RoboDK station: Simulation & programs.rdk

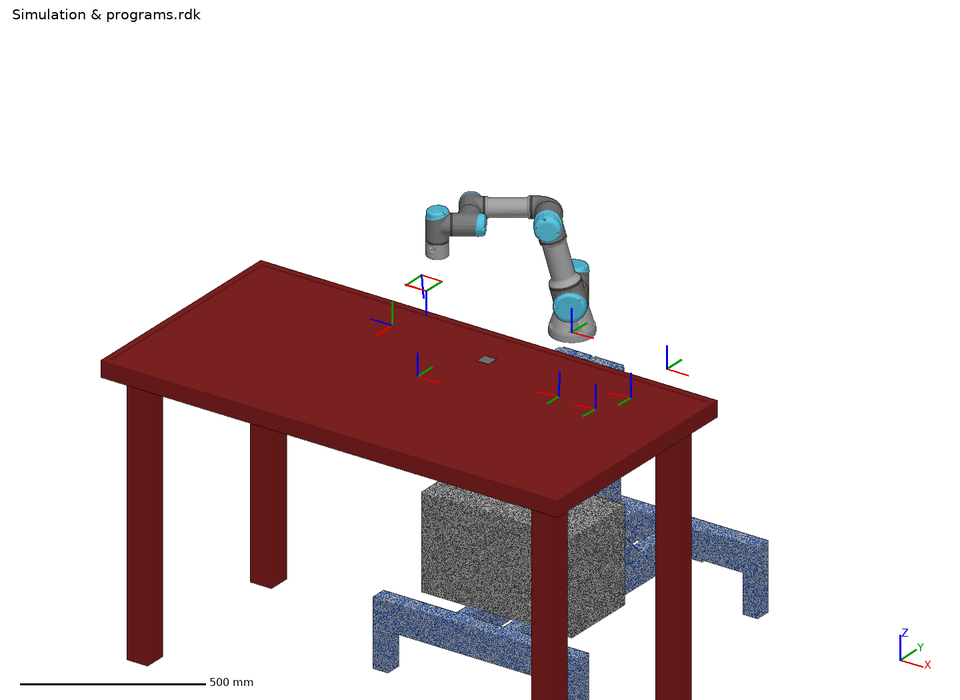
[picture v0: the station drawn from its stored meshes, robots at their saved joint values, targets as dots, program paths as lines]
Station Simulacion_3e (saved by RoboDK 5.6.3). Poses are relative to the parent item; angles as X-Y-Z fixed-axis rotations.
Station parameters (name, value as stored): RECORD_READY, 1, RECORD_STOP, 0, RECORD_ACKNOWLEDGE, 1, RECORD_ROBOT, 1
  - frame UR3e Base at (0, 0, 0) mm
    - robot UR3e: 6 axes, payload 3 kg, reach 500 mm, repeatability 0.03 mm, weight 11 kg
        modified DH rows (alpha deg, a mm, theta deg, d mm): 0, 0, 0, 151.9; 90, 0, 180, 0; 0, 243.55, 0, 0; 0, 213.2, 0, 131.05; -90, 0, 0, 85.35; 90, 0, 180, 92.1
        joint limits [-360, -360, -360, -360, -360, -360] to [360, 360, 360, 360, 360, 360]; home [90, -90, 90, -90, -90, 0]; saved at [32.842, -75.693, 77.295, -91.601, -89.995, -57.158]
      - frame Frame_Camara_1 at (9.13, -59.06, 41.13) mm, rotated rx 2.97 ry 2.34 rz -176.88 deg
        - camera CamaraBrazo
      - tool Gripper 2, TCP at (0, -50, 90) mm
      - frame Frame 8 at (0, -50, 90) mm
    - frame huevo_0 at (365.18, -244.95, 4.03) mm, rotated rx 5.66 ry 2.48 rz -173.5 deg
    - frame huevo_1 at (340.38, -375.16, 14.87) mm, rotated rx 5.66 ry 2.48 rz -173.5 deg
    - frame huevo_2 at (204.36, -351.92, 5.32) mm, rotated rx 5.66 ry 2.48 rz -173.5 deg
  - object mesaUR v1 at (0, 0, -110) mm, rotated rx 0 ry 0 rz -90 deg, size 1282 x 1503 x 903.8 mm
  - frame Frame_Tablero at (-200.86, -439.4, -14.21) mm
    - object Checkerboard at (0, 0, 0) mm, size 148.6 x 105 x 0 mm, geometry from Checkerboard.png
  - frame Frame_Aruco_20 at (340, -40, 0) mm
    - object aruco-20 at (-450, -250, 0) mm, size 37.9 x 37.9 x 0 mm, geometry from aruco-20.png
  - object Huevo at (-87.8, -330.3, 0) mm, rotated rx 0 ry 0 rz 60 deg, size 44.9 x 57 x 45 mm, geometry from Huevo.STEP
  - object Huevo at (10, -320, 0) mm, rotated rx 0 ry 0 rz 140 deg, size 44.9 x 57 x 45 mm, geometry from Huevo.STEP
  - object Huevo at (400, -90, 0) mm, rotated rx 0 ry 0 rz -15 deg, size 44.9 x 57 x 45 mm, geometry from Huevo.STEP
  - Python program Hand-Eye acquisition (listed below)
  - Python program Hand-Eye calibration (listed below)
  - Python program Hand-Eye acquisition Aruco (listed below)
  - Python program Tomar Una Foto (listed below)
  - Python program Pos (listed below)
  - frame PrePallet at (-230.35, -354.58, 199.88) mm, rotated rx -179.99 ry 0 rz 179.99 deg
  - Python program USB (listed below)
  - Python program TestMQTT (listed below)
  - frame inicioPallet at (-350.36, -344.58, 59.9) mm, rotated rx 90 ry 0 rz -90 deg
  - Python program Pos2 (listed below)

--- Python program Hand-Eye acquisition ---
# Type help("robolink") or help("robodk") for more information
# Press F5 to run the script
# Documentation: https://robodk.com/doc/en/RoboDK-API.html
# Reference:     https://robodk.com/doc/en/PythonAPI/index.html
#
# Utility script to perform hand-eye calibration on a 2D camera.
# This script can be use for eye-in-hand or eye-to-hand calibrations.
# Dynamically record the robot pose and save the camera image on disk for later processing.
# This script is running in a separate thread and a main program request punctual recordings through an handshake.

from robodk import robolink  # RoboDK API
from robodk import robomath  # Robot toolbox

# Uncomment these lines to automatically install the dependencies using pip
# robolink.import_install('cv2', 'opencv-contrib-python==4.5.*')
# robolink.import_install('numpy')
import cv2 as cv
import numpy as np
from pathlib import Path
import json
from enum import Enum
import time


#--------------------------------------
# This script supports RoboDK virtual/simulated cameras, and USB devices (as supported by OpenCV)
# You can add your own implementation to retrieve images from any camera, such as a Cognex Insight, SICK, etc.
class CameraTypes(Enum):
    ROBODK_SIMULATED = 1
    OPENCV_USB = 0


RECORD_ROBOT = True  # Record the robot pose on disk
RECORD_CAMERA = True  # Record the camera image on disk
RECORD_FOLDER = 'Calibracion Hand - Eye Camara'  # Default folder to save recordings, relative to the station folder

CAMERA_TYPE = CameraTypes.OPENCV_USB  # Camera type to be used
CAMERA_ROBODK_NAME = 'My Camera'  # [Optional] Default name to use for the RoboDK camera
ROBOT_NAME = 'UR3e'  # [Optional] Default name to use for the robot

# Station variables shared with the main program to interact with this script
RECORD_READY = 'RECORD_READY'  # Set this true in the main program when the robot is in position and the the script is allowed to record the robot and the image
RECORD_ACKNOWLEDGE = 'RECORD_ACKNOWLEDGE'  # Set this true in this script when the record is complete
RECORD_STOP = 'RECORD_STOP'  # Request to stop the script by the main program


#--------------------------------------
def get_robot(RDK: robolink.Robolink, robot_name: str):

    # Retrieve the robot
    robot_item = None
    if robot_name:
        robot_item = RDK.Item(robot_name, robolink.ITEM_TYPE_ROBOT)
        if not robot_item.Valid():
            robot_name = ''

    if not robot_name:
        robot_item = RDK.ItemUserPick("Select the robot for hand-eye", robolink.ITEM_TYPE_ROBOT)
        if not robot_item.Valid():
            raise

    return robot_item


def get_camera_handle(camera_type: CameraTypes, camera_name: str, RDK: robolink.Robolink):

    if camera_type == CameraTypes.ROBODK_SIMULATED:

        # Retrieve the RoboDK camera by name
        camera_item = None
        if camera_name:
            camera_item = RDK.Item(camera_name, robolink.ITEM_TYPE_CAMERA)
            if not camera_item.Valid():
                camera_name = ''

        if not camera_name:
            camera_item = RDK.ItemUserPick("Select the camera for hand-eye", robolink.ITEM_TYPE_CAMERA)
            if not camera_item.Valid():
                raise

        # Ensure the preview window in RoboDK is open
        if camera_item.setParam('Open') != '1':
            camera_item.setParam('Open', 1)
            robomath.pause(0.1)

        return camera_item

    elif camera_type == CameraTypes.OPENCV_USB:
        return cv.VideoCapture(0, cv.CAP_ANY)  # More information on supported devices here: https://docs.opencv.org/4.x/d8/dfe/classcv_1_1VideoCapture.html#aabce0d83aa0da9af802455e8cf5fd181

    return None


def record_camera(camera_type: CameraTypes, camera_handle, filename: str):
    if camera_type == CameraTypes.ROBODK_SIMULATED:
        record_robodk_camera(filename, camera_handle)

    elif camera_type == CameraTypes.OPENCV_USB:
        record_opencv_camera(filename, camera_handle)


def record_robodk_camera(filename: str, camera_item: robolink.Item):

    # Retrieve the image by socket
    bytes_img = camera_item.RDK().Cam2D_Snapshot('', camera_item)
    nparr = np.frombuffer(bytes_img, np.uint8)
    img = cv.imdecode(nparr, cv.IMREAD_COLOR)

    # Save the image on disk as a grayscale image
    cv.imwrite(filename, cv.cvtColor(img, cv.COLOR_RGB2GRAY))


def record_opencv_camera(filename: str, capture: cv.VideoCapture(0)):

    capture.set(3, 1280)  # Ancho
    capture.set(4, 720)

    # Retrieve image
    success, img = capture.read()
    if not success:
        raise



    # Save the image on disk as a grayscale image
    cv.imwrite(filename, cv.cvtColor(img, cv.COLOR_RGB2GRAY))


def record_robot(robot_item: robolink.Item, filename: str):

    # Retrieve the required information for hand-eye
    robot_data = {}
    robot_data['joints'] = robot_item.Joints().tolist()
    robot_data['pose_flange'] = robomath.Pose_2_TxyzRxyz(robot_item.SolveFK(robot_item.Joints()))

    # Save it on disk as a JSON
    # You can also provide another format, like YAML
    with open(filename, 'w') as f:
        json.dump(robot_data, f, indent=2)


def runmain():

    RDK = robolink.Robolink()

    # Retrieve the camera and robot
    camera_handle = get_camera_handle(CAMERA_TYPE, CAMERA_ROBODK_NAME, RDK)
    #print ("Camera name:" + camera_handle.Name())
    robot_item = get_robot(RDK, ROBOT_NAME)
    #print ("Robot name:" + robot_item.Name())

    # Retrieve the folder to save the data
    record_folder = Path(RDK.getParam(robolink.PATH_OPENSTATION)) / RECORD_FOLDER
    record_folder.mkdir(exist_ok=True, parents=True)
    print ("Folder ok")
    # This script does not delete the previous run if the folder is not empty
    # If the folder is not empty, retrieve the next ID
    id = 0
    ids = sorted([int(x.stem) for x in record_folder.glob('*.png') if x.stem.isdigit()])
    if ids:
        id = ids[-1] + 1

    # Start the main loop, and wait for requests
    RDK.setParam(RECORD_READY, 0)
    while True:
        time.sleep(0.01)

        # Read the requests set by the main program
        ready = int(RDK.getParam(RECORD_READY)) == 1
        stop = int(RDK.getParam(RECORD_STOP)) == 1
        if stop:

            break

        if not ready:

            continue



        # Process the requests
        if RECORD_CAMERA:
            img_filename = Path(f'{record_folder.as_posix()}/{id}.png')
            record_camera(CAMERA_TYPE, camera_handle, img_filename.as_posix())

        if RECORD_ROBOT:
            robot_filename = Path(f'{record_folder.as_posix()}/{id}.json')
            record_robot(robot_item, robot_filename.as_posix())

        id += 1

        print(img_filename)
        print(robot_filename)

        # Inform the main program that we have completed the request
        RDK.setParam(RECORD_ACKNOWLEDGE, 1)
        RDK.setParam(RECORD_READY, 0)




if __name__ == '__main__':
    runmain()

--- Python program Hand-Eye calibration ---
# Type help("robolink") or help("robodk") for more information
# Press F5 to run the script
# Documentation: https://robodk.com/doc/en/RoboDK-API.html
# Reference:     https://robodk.com/doc/en/PythonAPI/index.html
#
# Perform hand-eye calibration with recorded robot poses and 2D images from disk.
# - Requires at least 8 different poses at different orientations/distances of a chessboard or charucoboard.
# - Requires a calibrated camera (known intrinsic parameters, including distortion), which can also be performed from local images.
#
# You can find the board used in this example here:
# https://docs.opencv.org/4.x/charucoboard.png
#

from robodk import robolink  # RoboDK API
from robodk import robomath  # Robot toolbox
from robodk import robodialogs  # Dialogs

# Uncomment these lines to automatically install the dependencies using pip
# robolink.import_install('cv2', 'opencv-contrib-python==4.5.*')
# robolink.import_install('numpy')
import cv2 as cv
import numpy as np
import json
from pathlib import Path
from enum import Enum


#--------------------------------------
# This scripts supports chessboard (checkerboard) and ChAruCo board as calibration objects.
# You can add your own implementation (such as dot patterns).
class MarkerTypes(Enum):
    CHESSBOARD = 0
    CHARUCOBOARD = 1


# The camera intrinsic parameters can be performed with the same board as the Hand-eye
INTRINSIC_FOLDER = 'B:/Descargas/Simulacion 3e/Simulacion 3e/Calibracion Hand - Eye Camara'  # Default folder to load images for the camera calibration, relative to the station folder
HANDEYE_FOLDER = 'B:/Descargas/Simulacion 3e/Simulacion 3e/Calibracion Hand - Eye Camara'
# Camera intrinsic calibration board parameters
# You can find this chessboard here: https://docs.opencv.org/4.x/charucoboard.png
INTRINSIC_BOARD_TYPE = MarkerTypes.CHESSBOARD
INTRINSIC_CHESS_SIZE = (11, 9)  # X/Y
INTRINSIC_SQUARE_SIZE = 18  # mm
INTRINSIC_MARKER_SIZE = 18 # mm

# Hand-eye calibration board parameters
# You can find this charucoboard here: https://docs.opencv.org/4.x/charucoboard.png
#HANDEYE_BOARD_TYPE = MarkerTypes.CHARUCOBOARD
HANDEYE_BOARD_TYPE = MarkerTypes.CHESSBOARD
HANDEYE_CHESS_SIZE = (11, 9)  # X/Y
HANDEYE_SQUARE_SIZE = 18 # mm
HANDEYE_MARKER_SIZE = 18 # mm


def pose_2_Rt(pose: robomath.Mat):
    """RoboDK pose to OpenCV pose"""
    pose_inv = pose.inv()
    R = np.array(pose_inv.Rot33())
    t = np.array(pose.Pos())
    return R, t


def Rt_2_pose(R, t):
    """OpenCV pose to RoboDK pose"""
    vx, vy, vz = R.tolist()

    cam_pose = robomath.eye(4)
    cam_pose.setPos([0, 0, 0])
    cam_pose.setVX(vx)
    cam_pose.setVY(vy)
    cam_pose.setVZ(vz)

    pose = cam_pose.inv()
    pose.setPos(t.tolist())

    return pose


def find_chessboard(img, mtx, dist, chess_size, squares_edge, refine=True, draw_img=None):
    """
    Detects a chessboard pattern in an image.
    """

    pattern = np.subtract(chess_size, (1, 1))  # number of corners

    # Prefer grayscale images
    _img = img
    if len(img.shape) > 2:
        _img = cv.cvtColor(img, cv.COLOR_RGB2GRAY)

    # Find the chessboard's corners
    success, corners = cv.findChessboardCorners(_img, pattern)
    if not success:
        raise Exception("No chessboard found")

    # Refine
    if refine:
        criteria = (cv.TERM_CRITERIA_EPS + cv.TERM_CRITERIA_MAX_ITER, 30, 0.001)
        search_size = (11, 11)
        zero_size = (-1, -1)
        corners = cv.cornerSubPix(_img, corners, search_size, zero_size, criteria)

    if draw_img is not None:
        cv.drawChessboardCorners(draw_img, pattern, corners, success)

    # Find the camera pose. Only available with the camera matrix!
    if mtx is None or dist is None:
        return corners, None, None

    cb_corners = np.zeros((pattern[0] * pattern[1], 3), np.float32)
    cb_corners[:, :2] = np.mgrid[0:pattern[0], 0:pattern[1]].T.reshape(-1, 2) * squares_edge
    success, rvec, tvec = cv.solvePnP(cb_corners, corners, mtx, dist)
    if not success:
        raise Exception("No chessboard found")

    R_target2cam = cv.Rodrigues(rvec)[0]
    t_target2cam = tvec

    return corners, R_target2cam, t_target2cam


def find_charucoboard(img, mtx, dist, chess_size, squares_edge, markers_edge, predefined_dict=cv.aruco.DICT_6X6_100, draw_img=None) -> dict:
    """
    Detects a charuco board pattern in an image.
    """

    # Note that for chessboards, the pattern size is the number of "inner corners", while charucoboards are the number of chessboard squares

    # Charuco board and dictionary
    charuco_board = cv.aruco.CharucoBoard_create(chess_size[0], chess_size[1], squares_edge, markers_edge, cv.aruco.getPredefinedDictionary(predefined_dict))
    charuco_dict = charuco_board.dictionary

    # Find the markers first
    marker_corners, marker_ids, _ = cv.aruco.detectMarkers(img, charuco_dict, None, None, None, None)
    if marker_ids is None or len(marker_ids) < 1:
        raise Exception("No charucoboard found")

    # Then the charuco
    count, corners, ids = cv.aruco.interpolateCornersCharuco(marker_corners, marker_ids, img, charuco_board, None, None, mtx, dist, 2)  # mtx and dist are optional here
    if count < 1 or len(ids) < 1:
        raise Exception("No charucoboard found")

    if draw_img is not None:
        cv.aruco.drawDetectedCornersCharuco(draw_img, corners, ids)

    # Find the camera pose. Only available with the camera matrix!
    if mtx is None or dist is None:
        return corners, None, None

    success, rot_vec, trans_vec = cv.aruco.estimatePoseCharucoBoard(corners, ids, charuco_board, mtx, dist, None, None, False)  # mtx and dist are mandatory here
    if not success:
        raise Exception("Charucoboard pose not found")

    if draw_img is not None:
        cv.drawFrameAxes(draw_img, mtx, dist, rot_vec, trans_vec, max(1.5 * squares_edge, 5))

    R_target2cam = cv.Rodrigues(rot_vec)[0]

    return corners, R_target2cam, trans_vec


def calibrate_static(chessboard_images, board_type: MarkerTypes, chess_size, squares_edge: float, markers_edge: float, min_detect: int = -1, show_images=False):
    """
    Calibrate a camera with a chessboard or charucoboard pattern.
    """
    # Chessboard parameters
    pattern = np.subtract(chess_size, (1, 1))  # number of corners
    img_size = None

    # Find the chessboard corners
    img_corners = []

    if show_images:
        WDW_NAME = 'Chessboard'
        MAX_W, MAX_H = 640, 480
        cv.namedWindow(WDW_NAME, cv.WINDOW_NORMAL)

    for file, img in chessboard_images.items():
        # Ensure the image size is consistent
        if img_size is None:
            img_size = img.shape[:2]
        else:
            if img.shape[:2] != img_size:
                raise Exception('Camera resolution is not consistent across images!')

        # Find the chessboard corners
        draw_img = None
        if show_images:
            draw_img = cv.cvtColor(img, cv.COLOR_GRAY2RGB)
        try:
            if board_type == MarkerTypes.CHESSBOARD:
                corners, _, _ = find_chessboard(img, mtx=None, dist=None, chess_size=chess_size, squares_edge=squares_edge, draw_img=draw_img)
            else:
                corners, _, _ = find_charucoboard(img, mtx=None, dist=None, chess_size=chess_size, squares_edge=squares_edge, markers_edge=markers_edge, draw_img=draw_img)
        except:
            print(f'Unable to find chessboard in {file}!')
            continue

        if show_images:
            cv.imshow(WDW_NAME, draw_img)
            cv.resizeWindow(WDW_NAME, MAX_W, MAX_H)
            cv.waitKey(500)
        img_corners.append(corners)

        # Check if we processed enough images
        if min_detect > 0 and len(img_corners) >= min_detect:
            break

    if show_images:
        cv.destroyAllWindows()

    if len(img_corners) < 3 or min_detect > 0 and len(img_corners) < min_detect:
        raise Exception('Not enough detections!')

    # Calibrate the camera
    # Create a flat chessboard representation of the corners
    cb_corners = np.zeros((pattern[0] * pattern[1], 3), np.float32)
    cb_corners[:, :2] = np.mgrid[0:pattern[0], 0:pattern[1]].T.reshape(-1, 2) * squares_edge

    h, w = img_size
    rms_err, mtx, dist, rot_vecs, trans_vecs = cv.calibrateCamera([cb_corners for i in range(len(img_corners))], img_corners, (w, h), None, None)
    return mtx, dist, (w, h)


def calibrate_handeye(robot_poses, chessboard_images, camera_matrix, camera_distortion, board_type: MarkerTypes, chess_size, squares_edge: float, markers_edge: float, show_images=False):
    """
    Calibrate a camera mounted on a robot arm using a list of robot poses and a list of images for each pose.
    The robot pose should be at the flange (remove .PoseTool) unless you have a calibrated tool.
    """
    # https://docs.opencv.org/4.x/d9/d0c/group__calib3d.html#gaebfc1c9f7434196a374c382abf43439b

    # Rotation part extracted from the homogeneous matrix that transforms a point expressed in the gripper frame to the robot base frame (bTg).
    # This is a vector (vector<Mat>) that contains the rotation, (3x3) rotation matrices or (3x1) rotation vectors, for all the transformations from gripper frame to robot base frame.
    R_gripper2base_list = []

    # Translation part extracted from the homogeneous matrix that transforms a point expressed in the gripper frame to the robot base frame (bTg).
    # This is a vector (vector<Mat>) that contains the (3x1) translation vectors for all the transformations from gripper frame to robot base frame.
    t_gripper2base_list = []

    # Rotation part extracted from the homogeneous matrix that transforms a point expressed in the target frame to the camera frame (cTt).
    # This is a vector (vector<Mat>) that contains the rotation, (3x3) rotation matrices or (3x1) rotation vectors, for all the transformations from calibration target frame to camera frame.
    R_target2cam_list = []

    # Rotation part extracted from the homogeneous matrix that transforms a point expressed in the target frame to the camera frame (cTt).
    # This is a vector (vector<Mat>) that contains the (3x1) translation vectors for all the transformations from calibration target frame to camera frame.
    t_target2cam_list = []

    if show_images:
        WDW_NAME = 'Charucoboard'
        #WDW_NAME = 'Chessboard'
        MAX_W, MAX_H = 640, 480
        cv.namedWindow(WDW_NAME, cv.WINDOW_NORMAL)

    for i in chessboard_images.keys():
        robot_pose = robot_poses[i]
        image = chessboard_images[i]
        draw_img = None
        if show_images:
            draw_img = cv.cvtColor(image, cv.COLOR_GRAY2RGB)
        try:
            if board_type == MarkerTypes.CHESSBOARD:
                _, R_target2cam, t_target2cam = find_chessboard(image, camera_matrix, camera_distortion, chess_size, squares_edge, draw_img=draw_img)
            else:
                _, R_target2cam, t_target2cam = find_charucoboard(image, camera_matrix, camera_distortion, chess_size, squares_edge, markers_edge, draw_img=draw_img)
        except:
            print(f'Unable to find chessboard in {i}!')
            continue

        if show_images:
            cv.imshow(WDW_NAME, draw_img)
            cv.resizeWindow(WDW_NAME, MAX_W, MAX_H)
            cv.waitKey(500)

        R_target2cam_list.append(R_target2cam)
        t_target2cam_list.append(t_target2cam)

        R_gripper2base, t_gripper2base = pose_2_Rt(robot_pose)
        R_gripper2base_list.append(R_gripper2base)
        t_gripper2base_list.append(t_gripper2base)

    if show_images:
        cv.destroyAllWindows()

    R_cam2gripper, t_cam2gripper = cv.calibrateHandEye(R_gripper2base_list, t_gripper2base_list, R_target2cam_list, t_target2cam_list)
    return Rt_2_pose(R_cam2gripper, t_cam2gripper)


def runmain():
    #------------------------------------------------------
    # Calibrate the camera intrinsic parameters
    # 1. Print a chessboard, measure it using a caliper
    # 2. Mount the camera statically, take a series of images of the chessboard at different distance, orientation, offset, etc.
    # 3. Calibrate the camera using the images (can be done offline)
    #
    #
    # Calibrate the camera location (hand-eye)
    # 4. Create a robot program in RoboDK that moves the robot around a static chessboard at different distance, orientation, offset, etc.
    # 5. At each position, record the robot pose (robot.Pose(), or robot.Joints() even) and take a screenshot with the camera
    # 6. Use the robot poses and the images to calibrate the camera location
    #
    #
    # Good to know
    # - You can retrieve the camera image live with OpenCV using cv.VideoCapture(0, cv.CAP_DSHOW)
    # - You can load/save images with OpenCV using cv.imread(filename) and cv.imwrite(filename, img)
    # - You can save your calibrated camera parameters with JSON, i.e. print(json.dumps({"mtx":mtx, "dist":dist}))
    #
    #------------------------------------------------------

    RDK = robolink.Robolink()

    #------------------------------------------------------
    # Calibrate a camera using local images of chessboards, retrieves the camera intrinsic parameters
    # Get the input folder
    intrinsic_folder = Path(RDK.getParam(robolink.PATH_OPENSTATION)) / INTRINSIC_FOLDER
    if not intrinsic_folder.exists():
        intrinsic_folder = robodialogs.getSaveFolder(intrinsic_folder.as_posix(), 'Select the directory containing the images (.png) for the camera intrinsic calibration')
        if not intrinsic_folder:
            raise
        intrinsic_folder = Path(intrinsic_folder)

    # Retrieve the images
    image_files = sorted(intrinsic_folder.glob('*.png'))
    images = {int(image_file.stem): cv.imread(image_file.as_posix(), cv.IMREAD_GRAYSCALE) for image_file in image_files}

    # Perform the image calibration
    mtx, dist, size = calibrate_static(images, INTRINSIC_BOARD_TYPE, INTRINSIC_CHESS_SIZE, INTRINSIC_SQUARE_SIZE, INTRINSIC_MARKER_SIZE, min_detect=-1)
    print(f'Camera matrix:\n{mtx}\n')
    print(f'Distortion coefficient:\n{dist}\n')
    print(f'Camera resolution:\n{size}\n')

    #------------------------------------------------------
    # Load images and robot poses to calibrate hand-eye camera
    # Get the input folder
    handeye_folder = Path(RDK.getParam(robolink.PATH_OPENSTATION)) / HANDEYE_FOLDER
    if not handeye_folder.exists():
        handeye_folder = robodialogs.getSaveFolder('Select the directory of the images (.png) and robot poses (.json) for hand-eye calibration')
        if not handeye_folder:
            raise
        handeye_folder = Path(handeye_folder)

    # Retrieve the images and robot poses
    image_files = sorted(handeye_folder.glob('*.png'))
    robot_files = sorted(handeye_folder.glob('*.json'))

    images, poses, joints = {}, {}, {}
    for image_file, robot_file in zip(image_files, robot_files):
        if int(image_file.stem) != int(robot_file.stem):
            raise

        id = int(image_file.stem)

        image = cv.imread(image_file.as_posix(), cv.IMREAD_GRAYSCALE)
        images[id] = image

        with open(robot_file.as_posix(), 'r') as f:
            robot_data = json.load(f)
            joints[id] = robot_data['joints']
            poses[id] = robomath.TxyzRxyz_2_Pose(robot_data['pose_flange'])



    # Perform hand-eye calibration
    camera_pose = calibrate_handeye(poses, images, mtx, dist, HANDEYE_BOARD_TYPE, HANDEYE_CHESS_SIZE, HANDEYE_SQUARE_SIZE, HANDEYE_MARKER_SIZE)



    print(f'Camera pose (wrt to the robot flange):\n{camera_pose}')
    F_C = robomath.Pose_2_UR(camera_pose)
    F_C = np.array(F_C)
    F_C = F_C.tolist()
    ruta_F_C = "B:/Descargas/Simulacion 3e/Simulacion 3e/Matriz_F_C.json"


    mtx = mtx.tolist()
    dist = dist.tolist()
    calibracion = {'F_C':F_C, 'mtx':mtx , 'dist':dist}

    with open(ruta_F_C, 'w') as f:
        json.dump(calibracion, f)
    RDK.ShowMessage('Hand-Eye location:\n' + str(camera_pose))












    #------------------------------------------------------
    # In RoboDK, set the camera location wrt to the robot flange at that calibrated hand-eye location (use a .tool)
    tool = RDK.ItemUserPick('Select the "eye" tool to calibrate', RDK.ItemList(robolink.ITEM_TYPE_TOOL))

    if tool.Valid():
        tool.setPoseTool(camera_pose)




if __name__ == '__main__':
    runmain()

--- Python program Hand-Eye acquisition Aruco ---
# Type help("robolink") or help("robodk") for more information
# Press F5 to run the script
# Documentation: https://robodk.com/doc/en/RoboDK-API.html
# Reference:     https://robodk.com/doc/en/PythonAPI/index.html
#
# Utility script to perform hand-eye calibration on a 2D camera.
# This script can be use for eye-in-hand or eye-to-hand calibrations.
# Dynamically record the robot pose and save the camera image on disk for later processing.
# This script is running in a separate thread and a main program request punctual recordings through an handshake.

from robodk import robolink  # RoboDK API
from robodk import robomath  # Robot toolbox

# Uncomment these lines to automatically install the dependencies using pip
# robolink.import_install('cv2', 'opencv-contrib-python==4.5.*')
# robolink.import_install('numpy')
import cv2 as cv
import numpy as np
from pathlib import Path
import json
from enum import Enum
import time


#--------------------------------------
# This script supports RoboDK virtual/simulated cameras, and USB devices (as supported by OpenCV)
# You can add your own implementation to retrieve images from any camera, such as a Cognex Insight, SICK, etc.
class CameraTypes(Enum):
    ROBODK_SIMULATED = 0
    OPENCV_USB = 1


RECORD_ROBOT = True  # Record the robot pose on disk
RECORD_CAMERA = True  # Record the camera image on disk
RECORD_FOLDER = 'Hand-Eye-Data'  # Default folder to save recordings, relative to the station folder

CAMERA_TYPE = CameraTypes.ROBODK_SIMULATED  # Camera type to be used
CAMERA_ROBODK_NAME = 'My Camera'  # [Optional] Default name to use for the RoboDK camera
ROBOT_NAME = 'UR3e'  # [Optional] Default name to use for the robot

# Station variables shared with the main program to interact with this script
RECORD_READY = 'RECORD_READY'  # Set this true in the main program when the robot is in position and the the script is allowed to record the robot and the image
RECORD_ACKNOWLEDGE = 'RECORD_ACKNOWLEDGE'  # Set this true in this script when the record is complete
RECORD_STOP = 'RECORD_STOP'  # Request to stop the script by the main program


#--------------------------------------
def get_robot(RDK: robolink.Robolink, robot_name: str):

    # Retrieve the robot
    robot_item = None
    if robot_name:
        robot_item = RDK.Item(robot_name, robolink.ITEM_TYPE_ROBOT)
        if not robot_item.Valid():
            robot_name = ''

    if not robot_name:
        robot_item = RDK.ItemUserPick("Select the robot for hand-eye", robolink.ITEM_TYPE_ROBOT)
        if not robot_item.Valid():
            raise

    return robot_item


def get_camera_handle(camera_type: CameraTypes, camera_name: str, RDK: robolink.Robolink):

    if camera_type == CameraTypes.ROBODK_SIMULATED:

        # Retrieve the RoboDK camera by name
        camera_item = None
        if camera_name:
            camera_item = RDK.Item(camera_name, robolink.ITEM_TYPE_CAMERA)
            if not camera_item.Valid():
                camera_name = ''

        if not camera_name:
            camera_item = RDK.ItemUserPick("Select the camera for hand-eye", robolink.ITEM_TYPE_CAMERA)
            if not camera_item.Valid():
                raise

        # Ensure the preview window in RoboDK is open
        if camera_item.setParam('Open') != '1':
            camera_item.setParam('Open', 1)
            robomath.pause(0.1)

        return camera_item

    elif camera_type == CameraTypes.OPENCV_USB:
        return cv.VideoCapture(0, cv.CAP_ANY)  # More information on supported devices here: https://docs.opencv.org/4.x/d8/dfe/classcv_1_1VideoCapture.html#aabce0d83aa0da9af802455e8cf5fd181

    return None


def record_camera(camera_type: CameraTypes, camera_handle, filename: str):
    if camera_type == CameraTypes.ROBODK_SIMULATED:
        record_robodk_camera(filename, camera_handle)

    elif camera_type == CameraTypes.OPENCV_USB:
        record_opencv_camera(filename, camera_handle)


def record_robodk_camera(filename: str, camera_item: robolink.Item):

    # Retrieve the image by socket
    bytes_img = camera_item.RDK().Cam2D_Snapshot('', camera_item)
    nparr = np.frombuffer(bytes_img, np.uint8)
    img = cv.imdecode(nparr, cv.IMREAD_COLOR)

    # Save the image on disk as a grayscale image
    cv.imwrite(filename, img)


def record_opencv_camera(filename: str, capture: cv.VideoCapture):

    capture.set(3, 1280)  # Ancho
    capture.set(4, 720)

    # Retrieve image
    success, img = capture.read()
    if not success:
        raise

    # Save the image on disk as a grayscale image
    cv.imwrite(filename, img)


def record_robot(robot_item: robolink.Item, filename: str):

    # Retrieve the required information for hand-eye
    robot_data = {}
    robot_data['joints'] = robot_item.Joints().tolist()
    robot_data['pose_flange'] = robomath.Pose_2_TxyzRxyz(robot_item.SolveFK(robot_item.Joints()))

    # Save it on disk as a JSON
    # You can also provide another format, like YAML
    with open(filename, 'w') as f:
        json.dump(robot_data, f, indent=2)


def runmain():

    RDK = robolink.Robolink()

    # Retrieve the camera and robot
    camera_handle = get_camera_handle(CAMERA_TYPE, CAMERA_ROBODK_NAME, RDK)
    #print ("Camera name:" + camera_handle.Name())
    robot_item = get_robot(RDK, ROBOT_NAME)
    #print ("Robot name:" + robot_item.Name())

    # Retrieve the folder to save the data
    record_folder = Path(RDK.getParam(robolink.PATH_OPENSTATION)) / RECORD_FOLDER
    record_folder.mkdir(exist_ok=True, parents=True)
    print ("Folder ok")
    # This script does not delete the previous run if the folder is not empty
    # If the folder is not empty, retrieve the next ID
    id = 0
    ids = sorted([int(x.stem) for x in record_folder.glob('*.png') if x.stem.isdigit()])
    if ids:
        id = ids[-1] + 1

    # Start the main loop, and wait for requests
    RDK.setParam(RECORD_READY, 0)

    while True:
        time.sleep(0.01)

        # Read the requests set by the main program
        ready = int(RDK.getParam(RECORD_READY)) == 1
        stop = int(RDK.getParam(RECORD_STOP)) == 1
        if stop:
            break

        if not ready:
            continue

        # Process the requests
        if RECORD_CAMERA:
            img_filename = Path(f'{record_folder.as_posix()}/{id}.png')
            record_camera(CAMERA_TYPE, camera_handle, img_filename.as_posix())

        if RECORD_ROBOT:
            robot_filename = Path(f'{record_folder.as_posix()}/{id}.json')
            record_robot(robot_item, robot_filename.as_posix())

        id += 1

        print(img_filename)
        print(robot_filename)

        # Inform the main program that we have completed the request
        RDK.setParam(RECORD_ACKNOWLEDGE, 1)
        RDK.setParam(RECORD_READY, 0)


if __name__ == '__main__':
    runmain()

--- Python program Tomar Una Foto ---
from robodk import robolink
from robodk import robomath
RDK = robolink.Robolink()


from robodk import *
from robolink import *
import numpy as np

pause(2)
RECORD_READY = 'RECORD_READY'
RDK.setParam(RECORD_READY, 1)
pause(5)

--- Python program Pos ---
import cv2 as cv
import cv2.aruco as aruco
import numpy as np
import math
from scipy.spatial.transform import Rotation
from robodk import robolink
from robodk import robomath
RDK = robolink.Robolink()
from robodk import *
from robolink import *
import json
import os
import glob
from robolink import Robolink, ITEM_TYPE_FRAME
import paho.mqtt.client as mqtt

#hola boby

robot = RDK.Item('UR3e')
robot_frame = RDK.Item('UR3e Base')
frame = RDK.Item('Frame_Aruco_12')
frame_camara = RDK.Item('Frame_Camara_1')
gripper_tcp = RDK.Item('Gripper')
frame_inicio_pallet = RDK.Item('PrePallet')
arriba_pallet_inicio = RDK.Item('inicioPallet')
gripper_2 = RDK.Item('Gripper 2')
#robot.setTool(gripper_2)

frame_camara = RDK.Item('Frame_Camara_1')
ruta_F_C = "B:/Descargas/Simulacion 3e/Simulacion 3e/Matriz_F_C.json"
Mapeo_huevos = "B:/Descargas/Simulacion 3e/Simulacion 3e/Mapeo_Huevos.json"

with open(ruta_F_C, 'r') as f:
    calibracion = json.load(f)

with open(Mapeo_huevos, 'r') as f:
    mapeo= json.load(f)

pixeles_huevos = np.array(mapeo)



F_C = calibracion['F_C']
mtx = calibracion['mtx']
dist = calibracion['dist']
mtx = np.array(mtx)
dist = np.array(dist)
F_C = robomath.UR_2_Pose(F_C)


broker_address = "15.44.0.237" # Dirección del servidor MQTT
client = mqtt.Client("Antonio") # Nombre del cliente

global cap
cap = cv.VideoCapture(0)
cap.set(cv.CAP_PROP_FRAME_WIDTH, 1920)
cap.set(cv.CAP_PROP_FRAME_HEIGHT, 1080)










def pnp(corners):
    l = 40
    patron = np.array(
        [[0, l, 0], [l,l, 0], [l, 0, 0], [0, 0, 0]], dtype=np.float32
    )
    rvec_arr = np.empty((0, 3, 1))
    tvec_arr = np.empty((0, 3, 1))
    for esquina in corners:
        _, rvec, tvec = cv.solvePnP(patron, esquina, mtx, dist)
        rvec_arr = np.concatenate((rvec_arr, [rvec]), axis=0)
        tvec_arr = np.concatenate((tvec_arr, [tvec]), axis=0)

    return rvec_arr, tvec_arr

def ordenar_ids(marker_IDs, marker_corners):
        if marker_IDs is not None:
            sorted_indices = np.argsort(marker_IDs, axis=0)
            corners_sorted = np.array(marker_corners)[sorted_indices.flatten()]
            ids_sorted = np.array(marker_IDs)[sorted_indices.flatten()]
            return ids_sorted, corners_sorted
        else:
            return None, None

def promedio(id, aruco):
    caracteristicas_por_id = {}
    for id, caract in zip(id, aruco):
        if id[0] not in caracteristicas_por_id:
            caracteristicas_por_id[id[0]] = []
        caracteristicas_por_id[id[0]].append(caract)

    for id, caract in caracteristicas_por_id.items():
        caract = np.array(caract)
        promedio = np.mean(caract, axis=0)

    return promedio

def CalcularXYZ(u, v, A, rvec, tvec):
    Cord_reales = np.empty((0, 3, 1))

    for rot, tras in zip(rvec, tvec):
        uv = np.float64([[u, v, 1]]).T
        R, _ = cv.Rodrigues(rot)
        Inv_R = np.linalg.inv(R)
        Izda = Inv_R.dot(np.linalg.inv(A).dot(uv))
        Drch = Inv_R.dot(tras)
        s = -45 + Drch[2][0] / Izda[2][0]
        XYZ = Inv_R.dot(s * np.linalg.inv(A).dot(uv) - tras)
        Cord_reales = np.concatenate((Cord_reales, [XYZ]), axis=0)
    return Cord_reales

def medir_angulo_huevo(th):
    contornos , jerarquia = cv.findContours(th , cv.RETR_EXTERNAL , cv.CHAIN_APPROX_NONE)
    if len(contornos) != 0:

        for contorno in contornos:
            momento = cv.moments(contorno)
            if momento["m00"]>170000: #Limita el tamaño de los objetos que detecta
                #print(momento["m00"])
                elipse = cv.fitEllipse(contorno)
                centro , ejes , angulo = elipse

                centro = [int(centro[0]) , int(centro[1])]
                centroP = [centro[0] + 100 , centro[1] + 100]

                longitud = 100
                anguloP = angulo + 90


                x_extremo = int(centro[0] + longitud * np.cos(np.radians(angulo)))
                y_extremo = int(centro[1] + longitud * np.sin(np.radians(angulo)))

                x_1 = int(centro[0] + longitud * np.cos(np.radians(anguloP)))
                y_1 = int(centro[1] + longitud * np.sin(np.radians(anguloP)))

                angulo_horizontal = np.degrees(np.arctan2(y_1 - centro[1], x_1 - centro[0]))
                angulo_horizontal3 = (90 - anguloP) % 360




        return angulo_horizontal3 , centro



def pos_juntas(all_solutions):
    joints = []
    for j in all_solutions:
        conf_RLF = robot.JointsConfig(j).list()
        rear  = conf_RLF[0]
        lower = conf_RLF[1]
        flip  = conf_RLF[2]
        if rear == 1 and lower == 0 and flip == 1:
            joints = j
            break
    return joints
def configuraciones(pose):
    configuraciones = robot.SolveIK_All(pose, robot.PoseTool())
    return configuraciones

def control_angulo_RDK():
    CAM_NAME = 'CamaraBrazo'
    CAM_PARAMS = 'SIZE=1280x720'
    WINDOW_NAME = 'My Camera Feed'
    WINDOW_NAME_BW = 'My Camera BW'


    cam_item = RDK.Item(CAM_NAME, robolink.ITEM_TYPE_CAMERA)
    if not cam_item.Valid():
        cam_item = RDK.Cam2D_Add(RDK.AddFrame(CAM_NAME + ' Frame'), CAM_PARAMS)
        cam_item.setName(CAM_NAME)
    cam_item.setParam('Open', 1)

    angulo_referencia = 360
    while cam_item.setParam('isOpen') == '1':
        img_socket = None
        bytes_img = RDK.Cam2D_Snapshot('', cam_item)
        if isinstance(bytes_img, bytes) and bytes_img != b'':
            nparr = np.frombuffer(bytes_img, np.uint8)
            img_socket = cv.imdecode(nparr, cv.IMREAD_COLOR)
        if img_socket is None:
            break

        grayImage = cv.cvtColor(img_socket, cv.COLOR_BGR2GRAY)
        ret, img_bw = cv.threshold(grayImage, 200, 255, cv.THRESH_BINARY)
        #th = cv.bitwise_not(img_bw)
        angulo, centro  = medir_angulo_huevo(img_bw, img)


        error = angulo-angulo_referencia
        if angulo < 190 or angulo >350:
            #error = 200
            pause(1)
            return('Orientacion correcta')
        else:
            pos_nueva = robot.Pose()*rotz((error*pi/180)*0.2)
            pos_nueva = pos_juntas(configuraciones( pos_nueva))
            robot.MoveJ(pos_nueva)

        key = cv.waitKey(1)
        if key == 27:
            break  # User pressed ESC, exit

    cv.destroyAllWindows()
    RDK.Cam2D_Close(cam_item)

def control_angulo_OPENC_CV():
    angulo_referencia = 360
    while cap:
        ret, frame = cap.read()

        grayImage = cv.cvtColor(frame, cv.COLOR_BGR2GRAY)
        ret, img_bw = cv.threshold(grayImage, 132, 200, cv.THRESH_BINARY)
        #th = cv.bitwise_not(img_bw)
        angulo, centro  = medir_angulo_huevo(img_bw)
        centro1 = [centro[0] + 100 , centro [1] + 100]
        cv.putText(frame, str(angulo), (50, 50), cv.FONT_HERSHEY_SIMPLEX,2, (255, 0, 0), thickness=2)

        cv.imshow("Th" , img_bw)
        cv.imshow("fr" , frame)

        error = angulo-angulo_referencia
        if angulo < 187 or angulo >343:
              return('Orientacion correcta')
        else:
            pos_nueva = robot.Pose()*rotz((error*pi/180)*0.1)
            pos_nueva = pos_juntas(configuraciones( pos_nueva))
            robot.MoveJ(pos_nueva)
            print(angulo)

        if cv.waitKey(1) & 0xFF == ord('q'):
            break
    cap.release()
    cv.destroyAllWindows()


def controlador_posicion_RDK():
    CAM_NAME = 'CamaraBrazo'
    CAM_PARAMS = 'SIZE=1280x720'
    WINDOW_NAME = 'My Camera Feed'
    WINDOW_NAME_BW = 'My Camera BW'


    cam_item = RDK.Item(CAM_NAME, robolink.ITEM_TYPE_CAMERA)
    if not cam_item.Valid():
        cam_item = RDK.Cam2D_Add(RDK.AddFrame(CAM_NAME + ' Frame'), CAM_PARAMS)
        cam_item.setName(CAM_NAME)
    cam_item.setParam('Open', 1)

    centro_referencia = [640, 360]
    centro_referencia = np.array(centro_referencia)
    ganancia = -0.1
    while cam_item.setParam('isOpen') == '1':
        img_socket = None
        bytes_img = RDK.Cam2D_Snapshot('', cam_item)
        if isinstance(bytes_img, bytes) and bytes_img != b'':
            nparr = np.frombuffer(bytes_img, np.uint8)
            img_socket = cv.imdecode(nparr, cv.IMREAD_COLOR)
        if img_socket is None:
            break

        grayImage = cv.cvtColor(img_socket, cv.COLOR_BGR2GRAY)
        ret, img_bw = cv.threshold(grayImage, 200, 255, cv.THRESH_BINARY)
        contornos, r = cv.findContours(img_bw, cv.RETR_TREE, cv.CHAIN_APPROX_SIMPLE)
        #th = cv.bitwise_not(img_bw)
        for contorno in contornos:
            momento = cv.moments(contorno)


            if momento["m00"] > 27000 :
                cx = int(momento["m10"] / momento["m00"])
                cy = int(momento["m01"] / momento["m00"])


        centro = np.array([cx, cy])

        norma = np.linalg.norm(centro_referencia - centro)


        e_x_g = (centro_referencia[0]- cx )*ganancia
        e_y_g = (centro_referencia[1] - cy)*ganancia


        if norma > 20:
            pos_new =robot.Pose()*transl(e_x_g, e_y_g, 0)
            robot.MoveJ(pos_new)



        else:
            pause(1)

            return('1')

        cv.circle(img_socket, (cx, cy), 5, (255, 0,0), -1)
        cv.circle(img_socket, (centro_referencia[0], centro_referencia[1]), 5, (0, 255,0), -1)
        cv.imshow(WINDOW_NAME_BW, img_socket)


        key = cv.waitKey(1)
        if key == 27:
            break  # User pressed ESC, exit

    cv.destroyAllWindows()
    RDK.Cam2D_Close(cam_item)

def control_posicion_OPENC_CV():
    centro_referencia = [911 , 560]
    centro_referencia = np.array(centro_referencia)
    ganancia = 0.009
    while cap:
        ret, frame = cap.read()
        grayImage = cv.cvtColor(frame, cv.COLOR_BGR2GRAY)
        ret, img_bw = cv.threshold(grayImage, 132, 200, cv.THRESH_BINARY)
        cv.circle(frame, (centro_referencia[0], centro_referencia[1]), 5, (0, 255,0), -1)
        cv.circle(img_bw, (centro_referencia[0], centro_referencia[1]), 5, (0, 255,0), -1)
        #th = cv.bitwise_not(img_bw)
        contornos, r = cv.findContours(img_bw, cv.RETR_TREE, cv.CHAIN_APPROX_SIMPLE)
        for contorno in contornos:
            momento = cv.moments(contorno)
            if momento["m00"] > 170000 :
                cx = int(momento["m10"] / momento["m00"])
                cy = int(momento["m01"] / momento["m00"])
                print(cx, cy)
        centro = np.array([cx, cy])
        norma = np.linalg.norm(centro_referencia - centro)
        e_x_g = (centro_referencia[0]- cx )*ganancia
        e_y_g = (centro_referencia[1] - cy)*ganancia
        if norma > 8:
            pos_new =robot.Pose()*transl(e_x_g, e_y_g, 0)
            robot.MoveJ(pos_new)
            print(norma)
            return '1'
        else:
            print('Posicion corregida')
            #return('1')
        cv.circle(frame, (cx, cy), 5, (255, 0,0), -1)
        cv.circle(img_bw, (cx, cy), 5, (255, 0,0), -1)

        cv.imshow('1', frame)
        cv.imshow('2', img_bw)
        if cv.waitKey(1) & 0xFF == ord('q'):
            break
    cap.release()
    cv.destroyAllWindows()

def pallet_size(n, x_p, y_p):
    if n % x_p != 0:
        x = (n // x_p)+1
    else:
        x = n / x_p
    y = []
    for i in range(x):
        if n - y_p > 0:
            y.append(y_p)
        else:
            y.append(n % y_p)
        n = n - y_p
    return x,

def on_message(client, userdata, message):
    global mensaje_global
    mensaje_global = str(message.payload.decode("utf-8"))















ruta_carpeta = "B:/Descargas/Simulacion 3e/Simulacion 3e/Hand-Eye-Data"

archivos_json = sorted(glob.glob(os.path.join(ruta_carpeta, '*.json')))

imagenes = glob.glob(os.path.join(ruta_carpeta, '*.png'))

assert len(archivos_json) == len(imagenes), "La cantidad de archivos .json e imágenes no coincide"
mapa_aruco = np.empty([0,6])
mapa_id = np.empty([0,1])
for archivo_json, img, huevos_pix in zip(archivos_json, imagenes, pixeles_huevos):
    with open(archivo_json, 'r') as f:
        data = json.load(f)

    B_F = data["pose_flange"]
    B_F = robomath.TxyzRxyz_2_Pose(B_F)
    B_F = robomath.Mat(B_F)

    img = cv.imread(img)
    gray_frame = cv.cvtColor(img, cv.COLOR_BGR2GRAY)
    marker_dict = cv.aruco.getPredefinedDictionary(cv.aruco.DICT_ARUCO_ORIGINAL)
    param_markers = cv.aruco.DetectorParameters()
    detector = cv.aruco.ArucoDetector(marker_dict, param_markers)
    marker_corners, marker_IDs, _ = detector.detectMarkers(gray_frame)



    if marker_IDs is not None:


        marker_IDs, marker_corners =  ordenar_ids(marker_IDs, marker_corners)

        rvec_arr, tvec_arr = pnp(marker_corners)

        MTH_huevos = []
        for huevos_imagen in huevos_pix:
            cv.circle(img, huevos_imagen, 2, (255, 0, 0), 2)

            XYZ = CalcularXYZ(
            huevos_imagen[0], huevos_imagen[1], mtx, rvec_arr, tvec_arr
            )
            XYZ = XYZ[0]
            XYZ[-1, 0] = 23
            rotacion = np.eye(3)
            transformacion = np.eye(4)
            transformacion[:3, :3] = rotacion
            transformacion[:3, 3] = XYZ.flatten()
            MTH_huevos.append(transformacion)

        MTH_huevos = np.stack(MTH_huevos)

        pose_arucos = np.empty((0,6))
        ids_aruco = np.empty([0,1])
        for rot, tras, id in zip(rvec_arr, tvec_arr, marker_IDs):
            C_A_rot, _ = cv.Rodrigues(rot)
            C_A = np.eye(4)
            C_A[:3, :3] = C_A_rot
            C_A[:3, 3] = tras.flatten()
            C_A = robomath.Mat(C_A.tolist())
            C_A = robomath.Pose_2_UR(C_A)
            C_A = robomath.UR_2_Pose(C_A)



            B_A = B_F *F_C * C_A
            B_A = robomath.Pose_2_UR(B_A)



            B_A = np.array([B_A])
            pose_arucos = np.append(pose_arucos, B_A, axis=0)
            ids_aruco = np.append(ids_aruco, [id], axis = 0)
            cv.drawFrameAxes(img, mtx, dist, rot, tras, 30)

        mapa_aruco = np.vstack((mapa_aruco, pose_arucos))
        mapa_id = np.vstack((mapa_id, ids_aruco))

pos_aruco = promedio(mapa_id, mapa_aruco)

numero_huevos = 0
for huevo in MTH_huevos:

    huevo = robomath.Mat(huevo.tolist())
    B_A = UR_2_Pose(pos_aruco.tolist())
    B_H = B_A * huevo


    nombre_frame = 'huevo_' + str(numero_huevos)
    numero_huevos = numero_huevos + 1
    frame = RDK.AddFrame(nombre_frame)
    frame.setParent(robot_frame)
    frame.setPose(B_H)



frames = RDK.ItemList(ITEM_TYPE_FRAME)

frames_huevos = []
for frame in frames:
    if frame.Name().startswith('huevo_'):
        frames_huevos.append(RDK.Item(frame.Name()))


robot.MoveJ(robot.JointsHome())
mensaje_global = ''
dist_x = 0
aumento = 30#distancia entre centro bandeja
dist_bajar = 15
robot.setTool(gripper_2)

for frame_huevo in frames_huevos:
    pause(1)
    #-35
    #-65 lectura camara
    obj_H = frame_huevo.Pose()*rotx(pi)*transl(0, 0, -100)
    obj_H = pos_juntas(configuraciones(obj_H))
    robot.MoveJ(obj_H)
    pause(1)



    control_angulo_OPENC_CV()
    pause(1)
    control_posicion_OPENC_CV()
    arriba = robot.Pose()
    recoger = arriba*transl(0, 0, 10)
    robot.MoveL(recoger)
    pause(1)
    control_posicion_OPENC_CV()


    pause(1)

    arriba = robot.Pose()
    recoger = arriba*transl(0, 0, 65)#cambia
    robot.MoveL(recoger)
    pause(5)

    ## ######Cierra Gripper######
    client.connect(broker_address)
    client.subscribe("Terranator")
    client.publish("Terranator", "cerrar")
    while True:
        client.loop()
        client.on_message = on_message
        if mensaje_global == 'listo':
            print('1')
            mensaje_global = ''
            break
    # ######Gripper ya cerrado#####

    robot.MoveL(arriba)
    pause(1)
    pallet = frame_inicio_pallet.Pose()
    pallet = pos_juntas(configuraciones(pallet))
    robot.MoveJ(pallet)

    #pause(0.5)
    #pos_pallet = robot.Pose()* transl(0,-dist_bajar,0)
    #robot.MoveL(pos_pallet)
    #pause(0.5)
    #robot.MoveL(robot.Pose()* transl(0,dist_bajar,0))




  #  # #######Abre el gripper
    client.publish("Terranator", "abrir")
    while True:
        client.loop()
        client.on_message = on_message# Función que se ejecuta cuando se recibe un mensaje
        if mensaje_global == 'listo1':
            print('1')
            mensaje_global = ''
            break
    # ######Se confirma que ya esta abierto


robot.MoveJ(robot.JointsHome())

--- Python program USB ---
from robodk import robolink
from robodk import robomath

import cv2 as cv
import numpy as np
from pathlib import Path
import json
from enum import Enum
import time

RDK = robolink.Robolink()


RECORD_FOLDER = 'B:/Descargas/Simulacion 3e/Simulacion 3e/Hand-Eye-Data'
robot = RDK.Item('UR3e')


def runmain():
    cap = cv.VideoCapture(0)
    cap.set(cv.CAP_PROP_FRAME_WIDTH, 1920)
    cap.set(cv.CAP_PROP_FRAME_HEIGHT, 1080)
    RDK = robolink.Robolink()
    robot_item = robot
    record_folder = Path(RDK.getParam(robolink.PATH_OPENSTATION)) / RECORD_FOLDER
    record_folder.mkdir(exist_ok=True, parents=True)
    print ("Folder ok")
    ids = sorted([int(x.stem) for x in record_folder.glob('*.png') if x.stem.isdigit()])
    if ids:
        id = ids[-1] + 1

    else:
        id = 0

    while cap:
        time.sleep(0.01)
        ret, frame = cap.read()
        cv.imshow('Video de mi cámara', frame)
        if cv.waitKey(1) & 0xFF == ord('a'):
            RDK.setParam('RECORD_ROBOT', 1)
            img_filename = Path(f'{record_folder.as_posix()}/{id}.png')
            img_filename = str(img_filename)
            print(img_filename)
            cv.imwrite(img_filename, frame)
            robot_filename = Path(f'{record_folder.as_posix()}/{id}.json')
            robot_data = {}
            robot_data['joints'] = robot_item.Joints().tolist()
            robot_data['pose_flange'] = robomath.Pose_2_TxyzRxyz(robot_item.SolveFK(robot_item.Joints()))
            with open(robot_filename, 'w') as f:

                json.dump(robot_data, f, indent=2)

            id += 1


if __name__ == '__main__':
    runmain()

--- Python program TestMQTT ---
# Type help("robodk.robolink") or help("robodk.robomath") for more information
# Press F5 to run the script
# Documentation: https://robodk.com/doc/en/RoboDK-API.html
# Reference:     https://robodk.com/doc/en/PythonAPI/robodk.html
# Note: It is not required to keep a copy of this file, your Python script is saved with your RDK project

# You can also use the new version of the API:
from robodk import robolink    # RoboDK API
from robodk import robomath    # Robot toolbox
RDK = robolink.Robolink()

# Forward and backwards compatible use of the RoboDK API:
# Remove these 2 lines to follow python programming guidelines
from robodk import *      # RoboDK API
from robolink import *    # Robot toolbox
# Link to RoboDK
# RDK = Robolink()

import paho.mqtt.client as mqtt

# Función que se ejecuta cuando se recibe un mensaje
def on_message(client, userdata, message):
    print("Mensaje recibido: " + str(message.payload.decode("utf-8")))

# Configuración del cliente MQTT
broker_address = "10.25.66.214" # Dirección del servidor MQTT
client = mqtt.Client("Antonio") # Nombre del cliente
client.on_message = on_message # Función que se ejecuta cuando se recibe un mensaje
client.connect(broker_address) # Conexión al servidor MQTT
client.subscribe("Terranator") # Suscripción al tema "mi_tema"

# Envío de un mensaje
mensaje = "xddd"
client.publish("Terranator", mensaje)

# Bucle principal
while True:
    client.loop()
    # Realiza otras tareas aquí

--- Python program Pos2 ---
import cv2 as cv
import cv2.aruco as aruco
import numpy as np
import math
from scipy.spatial.transform import Rotation
from robodk import robolink
from robodk import robomath
RDK = robolink.Robolink()
from robodk import *
from robolink import *
import json
import os
import glob
from robolink import Robolink, ITEM_TYPE_FRAME
import paho.mqtt.client as mqtt


robot = RDK.Item('UR3e')
robot_frame = RDK.Item('UR3e Base')
frame = RDK.Item('Frame_Aruco_12')
frame_camara = RDK.Item('Frame_Camara_1')
gripper_tcp = RDK.Item('Gripper')
frame_inicio_pallet = RDK.Item('PrePallet')
arriba_pallet_inicio = RDK.Item('inicioPallet')
gripper_2 = RDK.Item('Gripper 2')
#robot.setTool(gripper_2)

frame_camara = RDK.Item('Frame_Camara_1')
ruta_F_C = "B:/Descargas/Simulacion 3e/Simulacion 3e/Matriz_F_C.json"
Mapeo_huevos = "B:/Descargas/Simulacion 3e/Simulacion 3e/Mapeo_Huevos.json"

with open(ruta_F_C, 'r') as f:
    calibracion = json.load(f)

with open(Mapeo_huevos, 'r') as f:
    mapeo= json.load(f)

pixeles_huevos = np.array(mapeo)

#camara
camara = 1 # Camara = 0; RoboDK, Camara = 1; openCV_USB

F_C = calibracion['F_C']
mtx = calibracion['mtx']
dist = calibracion['dist']
mtx = np.array(mtx)
dist = np.array(dist)
F_C = robomath.UR_2_Pose(F_C)


broker_address = "10.25.66.214" # Dirección del servidor MQTT
client = mqtt.Client("Diego") # Nombre del cliente

#global cap
#cap = cv.VideoCapture(0)
#cap.set(cv.CAP_PROP_FRAME_WIDTH, 1920)
#cap.set(cv.CAP_PROP_FRAME_HEIGHT, 1080)



def pnp(corners):
    l = 40
    patron = np.array(
        [[0, l, 0], [l,l, 0], [l, 0, 0], [0, 0, 0]], dtype=np.float32
    )
    rvec_arr = np.empty((0, 3, 1))
    tvec_arr = np.empty((0, 3, 1))
    for esquina in corners:
        _, rvec, tvec = cv.solvePnP(patron, esquina, mtx, dist)
        rvec_arr = np.concatenate((rvec_arr, [rvec]), axis=0)
        tvec_arr = np.concatenate((tvec_arr, [tvec]), axis=0)

    return rvec_arr, tvec_arr

def ordenar_ids(marker_IDs, marker_corners):
        if marker_IDs is not None:
            sorted_indices = np.argsort(marker_IDs, axis=0)
            corners_sorted = np.array(marker_corners)[sorted_indices.flatten()]
            ids_sorted = np.array(marker_IDs)[sorted_indices.flatten()]
            return ids_sorted, corners_sorted
        else:
            return None, None

def promedio(id, aruco):
    caracteristicas_por_id = {}
    for id, caract in zip(id, aruco):
        if id[0] not in caracteristicas_por_id:
            caracteristicas_por_id[id[0]] = []
        caracteristicas_por_id[id[0]].append(caract)

    for id, caract in caracteristicas_por_id.items():
        caract = np.array(caract)
        promedio = np.mean(caract, axis=0)

    return promedio

def CalcularXYZ(u, v, A, rvec, tvec):
    Cord_reales = np.empty((0, 3, 1))

    for rot, tras in zip(rvec, tvec):
        uv = np.float64([[u, v, 1]]).T
        R, _ = cv.Rodrigues(rot)
        Inv_R = np.linalg.inv(R)
        Izda = Inv_R.dot(np.linalg.inv(A).dot(uv))
        Drch = Inv_R.dot(tras)
        s = -45 + Drch[2][0] / Izda[2][0]
        XYZ = Inv_R.dot(s * np.linalg.inv(A).dot(uv) - tras)
        Cord_reales = np.concatenate((Cord_reales, [XYZ]), axis=0)
    return Cord_reales

def medir_angulo_huevo(th, img):
    contornos , jerarquia = cv.findContours(th , cv.RETR_EXTERNAL , cv.CHAIN_APPROX_NONE)
    if len(contornos) != 0:

        for contorno in contornos:
            momento = cv.moments(contorno)
            if momento["m00"] > 27000 : #Limita el tamaño de los objetos que detecta
                elipse = cv.fitEllipse(contorno)
                centro , ejes , angulo = elipse

                centro = [int(centro[0]) , int(centro[1])]
                centroP = [centro[0] + 100 , centro[1] + 100]

                longitud = 100
                anguloP = angulo + 90

                x_extremo = int(centro[0] + longitud * np.cos(np.radians(angulo)))
                y_extremo = int(centro[1] + longitud * np.sin(np.radians(angulo)))

                x_1 = int(centro[0] + longitud * np.cos(np.radians(anguloP)))
                y_1 = int(centro[1] + longitud * np.sin(np.radians(anguloP)))

                angulo_horizontal = np.degrees(np.arctan2(y_1 - centro[1], x_1 - centro[0]))
                angulo_horizontal3 = (90 - anguloP) % 360


        return angulo_horizontal3 , centro



def pos_juntas(all_solutions):
    joints = []
    for j in all_solutions:
        conf_RLF = robot.JointsConfig(j).list()
        rear  = conf_RLF[0]
        lower = conf_RLF[1]
        flip  = conf_RLF[2]
        if rear == 1 and lower == 0 and flip == 1:
            joints = j
            break
    return joints
def configuraciones(pose):
    configuraciones = robot.SolveIK_All(pose, robot.PoseTool())
    return configuraciones

def control_angulo_RDK():
    CAM_NAME = 'CamaraBrazo'
    CAM_PARAMS = 'SIZE=1280x720'
    WINDOW_NAME = 'My Camera Feed'
    WINDOW_NAME_BW = 'My Camera BW'


    cam_item = RDK.Item(CAM_NAME, robolink.ITEM_TYPE_CAMERA)
    if not cam_item.Valid():
        cam_item = RDK.Cam2D_Add(RDK.AddFrame(CAM_NAME + ' Frame'), CAM_PARAMS)
        cam_item.setName(CAM_NAME)
    cam_item.setParam('Open', 1)

    angulo_referencia = 360
    while cam_item.setParam('isOpen') == '1':
        img_socket = None
        bytes_img = RDK.Cam2D_Snapshot('', cam_item)
        if isinstance(bytes_img, bytes) and bytes_img != b'':
            nparr = np.frombuffer(bytes_img, np.uint8)
            img_socket = cv.imdecode(nparr, cv.IMREAD_COLOR)
        if img_socket is None:
            break

        grayImage = cv.cvtColor(img_socket, cv.COLOR_BGR2GRAY)
        ret, img_bw = cv.threshold(grayImage, 200, 255, cv.THRESH_BINARY)
        #th = cv.bitwise_not(img_bw)
        angulo, centro  = medir_angulo_huevo(img_bw, img)


        error = angulo-angulo_referencia
        if angulo < 190 or angulo >350:
            #error = 200
            pause(1)
            return('Orientacion correcta')
        else:
            pos_nueva = robot.Pose()*rotz((error*pi/180)*0.2)
            pos_nueva = pos_juntas(configuraciones( pos_nueva))
            robot.MoveJ(pos_nueva)

        key = cv.waitKey(1)
        if key == 27:
            break  # User pressed ESC, exit

    cv.destroyAllWindows()
    RDK.Cam2D_Close(cam_item)

def control_angulo_OPENC_CV():
    angulo_referencia = 360

    while cap:
        ret, frame = cap.read()

        grayImage = cv.cvtColor(frame, cv.COLOR_BGR2GRAY)
        ret, img_bw = cv.threshold(grayImage, 115, 255, cv.THRESH_BINARY)
        #th = cv.bitwise_not(img_bw)
        angulo, centro  = medir_angulo_huevo(img_bw, img)

        cv.imshow("Th" , img_bw)
        cv.imshow("fr" , frame)

        error = angulo-angulo_referencia
        if angulo < 190 or angulo >350:
             pause(1)
             return('Orientacion correcta')
        else:
            pos_nueva = robot.Pose()*rotz((error*pi/180)*0.1)
            pos_nueva = pos_juntas(configuraciones( pos_nueva))
            robot.MoveJ(pos_nueva)
            print(angulo)
        if cv.waitKey(1) & 0xFF == ord('q'):
            break
    cap.release()
    cv.destroyAllWindows()

def controlador_posicion_RDK():
    CAM_NAME = 'CamaraBrazo'
    CAM_PARAMS = 'SIZE=1280x720'
    WINDOW_NAME = 'My Camera Feed'
    WINDOW_NAME_BW = 'My Camera BW'


    cam_item = RDK.Item(CAM_NAME, robolink.ITEM_TYPE_CAMERA)
    if not cam_item.Valid():
        cam_item = RDK.Cam2D_Add(RDK.AddFrame(CAM_NAME + ' Frame'), CAM_PARAMS)
        cam_item.setName(CAM_NAME)
    cam_item.setParam('Open', 1)

    centro_referencia = [640, 360]
    centro_referencia = np.array(centro_referencia)
    ganancia = -0.1
    while cam_item.setParam('isOpen') == '1':
        img_socket = None
        bytes_img = RDK.Cam2D_Snapshot('', cam_item)
        if isinstance(bytes_img, bytes) and bytes_img != b'':
            nparr = np.frombuffer(bytes_img, np.uint8)
            img_socket = cv.imdecode(nparr, cv.IMREAD_COLOR)
        if img_socket is None:
            break

        grayImage = cv.cvtColor(img_socket, cv.COLOR_BGR2GRAY)
        ret, img_bw = cv.threshold(grayImage, 200, 255, cv.THRESH_BINARY)
        contornos, r = cv.findContours(img_bw, cv.RETR_TREE, cv.CHAIN_APPROX_SIMPLE)
        #th = cv.bitwise_not(img_bw)
        for contorno in contornos:
            momento = cv.moments(contorno)


            if momento["m00"] > 27000 :
                cx = int(momento["m10"] / momento["m00"])
                cy = int(momento["m01"] / momento["m00"])


        centro = np.array([cx, cy])

        norma = np.linalg.norm(centro_referencia - centro)


        e_x_g = (centro_referencia[0]- cx )*ganancia
        e_y_g = (centro_referencia[1] - cy)*ganancia


        if norma > 20:
            pos_new =robot.Pose()*transl(e_x_g, e_y_g, 0)
            robot.MoveJ(pos_new)



        else:
            pause(1)

            return('1')

        cv.circle(img_socket, (cx, cy), 5, (255, 0,0), -1)
        cv.circle(img_socket, (centro_referencia[0], centro_referencia[1]), 5, (0, 255,0), -1)
        cv.imshow(WINDOW_NAME_BW, img_socket)


        key = cv.waitKey(1)
        if key == 27:
            break  # User pressed ESC, exit

    cv.destroyAllWindows()
    RDK.Cam2D_Close(cam_item)

def control_posicion_OPENC_CV():
    centro_referencia = [960, 540]
    centro_referencia = np.array(centro_referencia)
    ganancia = 0.05
    while cap:
        ret, frame = cap.read()
        grayImage = cv.cvtColor(frame, cv.COLOR_BGR2GRAY)
        ret, img_bw = cv.threshold(grayImage, 200, 255, cv.THRESH_BINARY)
        th = cv.bitwise_not(img_bw)
        contornos, r = cv.findContours(th, cv.RETR_TREE, cv.CHAIN_APPROX_SIMPLE)
        for contorno in contornos:
            momento = cv.moments(contorno)
            if momento["m00"] > 50000 :
                cx = int(momento["m10"] / momento["m00"])
                cy = int(momento["m01"] / momento["m00"])
        centro = np.array([cx, cy])
        norma = np.linalg.norm(centro_referencia - centro)
        e_x_g = (centro_referencia[0]- cx )*ganancia
        e_y_g = (centro_referencia[1] - cy)*ganancia
        if norma > 20:
            pos_new =robot.Pose()*transl(e_x_g, e_y_g, 0)
            robot.MoveJ(pos_new)
            print(norma)
        else:
            pause(1)
            print('Posicion corregida')
            return('1')
        cv.circle(frame, (cx, cy), 5, (255, 0,0), -1)
        cv.circle(frame, (centro_referencia[0], centro_referencia[1]), 5, (0, 255,0), -1)
        cv.imshow('1', frame)
        if cv.waitKey(1) & 0xFF == ord('q'):
            break
    cap.release()
    cv.destroyAllWindows()

def pallet_size(n, x_p, y_p):
    if n % x_p != 0:
        x = (n // x_p)+1
    else:
        x = n / x_p
    y = []
    for i in range(x):
        if n - y_p > 0:
            y.append(y_p)
        else:
            y.append(n % y_p)
        n = n - y_p
    return x,

def on_message(client, userdata, message):
    global mensaje_global
    mensaje_global = str(message.payload.decode("utf-8"))




def maquina_estados():
    ruta_carpeta = "B:/Descargas/Simulacion 3e/Simulacion 3e/Hand-Eye-Data"
    archivos_json = sorted(glob.glob(os.path.join(ruta_carpeta, '*.json')))
    imagenes = glob.glob(os.path.join(ruta_carpeta, '*.png'))
    assert len(archivos_json) == len(imagenes),
    mapa_aruco = np.empty([0,6])
    mapa_id = np.empty([0,1])



for archivo_json, img, huevos_pix in zip(archivos_json, imagenes, pixeles_huevos):
    with open(archivo_json, 'r') as f:
        data = json.load(f)

    B_F = data["pose_flange"]
    B_F = robomath.TxyzRxyz_2_Pose(B_F)
    B_F = robomath.Mat(B_F)

    img = cv.imread(img)
    gray_frame = cv.cvtColor(img, cv.COLOR_BGR2GRAY)
    marker_dict = cv.aruco.getPredefinedDictionary(cv.aruco.DICT_ARUCO_ORIGINAL)
    param_markers = cv.aruco.DetectorParameters()
    detector = cv.aruco.ArucoDetector(marker_dict, param_markers)
    marker_corners, marker_IDs, _ = detector.detectMarkers(gray_frame)



    if marker_IDs is not None:


        marker_IDs, marker_corners =  ordenar_ids(marker_IDs, marker_corners)

        rvec_arr, tvec_arr = pnp(marker_corners)

        MTH_huevos = []
        for huevos_imagen in huevos_pix:
            cv.circle(img, huevos_imagen, 2, (255, 0, 0), 2)

            XYZ = CalcularXYZ(
            huevos_imagen[0], huevos_imagen[1], mtx, rvec_arr, tvec_arr
            )
            XYZ = XYZ[0]
            XYZ[-1, 0] = 23
            rotacion = np.eye(3)
            transformacion = np.eye(4)
            transformacion[:3, :3] = rotacion
            transformacion[:3, 3] = XYZ.flatten()
            MTH_huevos.append(transformacion)

        MTH_huevos = np.stack(MTH_huevos)

        pose_arucos = np.empty((0,6))
        ids_aruco = np.empty([0,1])
        for rot, tras, id in zip(rvec_arr, tvec_arr, marker_IDs):
            C_A_rot, _ = cv.Rodrigues(rot)
            C_A = np.eye(4)
            C_A[:3, :3] = C_A_rot
            C_A[:3, 3] = tras.flatten()
            C_A = robomath.Mat(C_A.tolist())
            C_A = robomath.Pose_2_UR(C_A)
            C_A = robomath.UR_2_Pose(C_A)



            B_A = B_F *F_C * C_A
            B_A = robomath.Pose_2_UR(B_A)



            B_A = np.array([B_A])
            pose_arucos = np.append(pose_arucos, B_A, axis=0)
            ids_aruco = np.append(ids_aruco, [id], axis = 0)
            cv.drawFrameAxes(img, mtx, dist, rot, tras, 30)

        mapa_aruco = np.vstack((mapa_aruco, pose_arucos))
        mapa_id = np.vstack((mapa_id, ids_aruco))

pos_aruco = promedio(mapa_id, mapa_aruco)

numero_huevos = 0
for huevo in MTH_huevos:

    huevo = robomath.Mat(huevo.tolist())
    B_A = UR_2_Pose(pos_aruco.tolist())
    B_H = B_A * huevo


    nombre_frame = 'huevo_' + str(numero_huevos)
    numero_huevos = numero_huevos + 1
    frame = RDK.AddFrame(nombre_frame)
    frame.setParent(robot_frame)
    frame.setPose(B_H)



frames = RDK.ItemList(ITEM_TYPE_FRAME)

frames_huevos = []
for frame in frames:
    if frame.Name().startswith('huevo_'):
        frames_huevos.append(RDK.Item(frame.Name()))


robot.MoveJ(robot.JointsHome())
mensaje_global = ''
dist_x = 0
aumento = 30#distancia entre centro bandeja
dist_bajar = 15
robot.setTool(gripper_2)

for frame_huevo in frames_huevos:
    pause(1)
    #-35
    #-65 lectura camara
    #print(robot.PoseTool())
    obj_H = invH(robot.Pose())*frame_huevo.Pose()
    print(frame_huevo.Pose())
    robot.MoveJ(frame_huevo.Pose()*rotx(pi))
    #obj_H = pos_juntas(configuraciones(obj_H))

    pause(1)
    #robot.MoveJ(robot.JointsHome())

    #if camara == 0:
        #orientacion = control_angulo_RDK()
        #controlador_posicion_RDK()

    #elif camara == 1:
        #control_angulo_OPENC_CV()
        #print("1")


    #arriba = robot.Pose()
    #recoger = arriba*transl(0, 0, 45)#cambia
    #robot.MoveL(recoger)
    #pause(1)

    ## ######Cierra Gripper######
    #client.connect(broker_address)
    #client.subscribe("Terranator")
    #client.publish("Terranator", "cerrar")
    #while True:
        #client.loop()
        #client.on_message = on_message
        #if mensaje_global == 'listo':
            #print('1')
            #mensaje_global = ''
            #break
    # ######Gripper ya cerrado#####

    #robot.MoveL(arriba)
    #pause(1)
    #pallet = frame_inicio_pallet.Pose()
    #pallet = pos_juntas(configuraciones(pallet))
    #robot.MoveJ(pallet)

    #pause(0.5)
    #pos_pallet = robot.Pose()* transl(0,-dist_bajar,0)
    #robot.MoveL(pos_pallet)
    #pause(0.5)
    #robot.MoveL(robot.Pose()* transl(0,dist_bajar,0))




  #  # #######Abre el gripper
   # client.publish("Terranator", "abrir")
    #while True:
        #client.loop()
        #client.on_message = on_message# Función que se ejecuta cuando se recibe un mensaje
        #if mensaje_global == 'listo1':
            #print('1')
            #mensaje_global = ''
            #break
    # ######Se confirma que ya esta abierto


robot.MoveJ(robot.JointsHome())
